// TIA Portal V15 export
// export: Created 2018-05-29T12:25:38.1552518Z, ExportSetting WithDefaults, DisplayName Totally Integrated Automation Portal, DisplayVersion V15, DisplayName STEP 7 Professional, DisplayVersion V15, DisplayName WinCC Professional, DisplayVersion V15, DisplayName TIA Portal Openness, DisplayVersion V15
FUNCTION_BLOCK "EM_I_OUT"   // FB1, STL
TITLE = EM_I_OUT_fc
{ S7_Optimized_Access := 'TRUE' }
VERSION : 0.1
// EM_I_OUT
// stored: AutoNumber true, UDAEnableTagReadback false
   VAR_INPUT
      sampletime : Real;   // the scantime of this EM/phase, used to increase timers
      em_id : Int;   // undefined - undefined
      Request : Int;   // undefined - undefined
      Command : Int;   // undefined - undefined
      Pressure_SP : REAL;   // undefined - undefined
      Pump_RUN : Bool;   // undefined - undefined
      Pump_QERR : BOOL;   // undefined - General Error
      Pump_EERR : BOOL;   // undefined - External Error
      FS01_PV : Bool;   // Flow Switch - Digital Measurement
      PIC01_PV : REAL;   // Pressure Controller - undefined
      PIC01_ERR : BOOL;   // Pressure Controller - undefined
      LT01_PV : Real;   // Level Transmitter (m) - undefined
      LT01_AHH : Bool;   // Level Transmitter (m) - undefined
      LT01_AH : Bool;   // Level Transmitter (m) - undefined
      LT01_AL : Bool;   // Level Transmitter (m) - undefined
      LT01_ALL : Bool;   // Level Transmitter (m) - undefined
      LT01_ERR : BOOL;   // Level Transmitter (m) - undefined
      XV_Bottom_OPN : BOOL;   // Automatic Bottom Valve - undefined
      XV_Bottom_CLS : BOOL;   // Automatic Bottom Valve - undefined
      XV_Bottom_MERR : BOOL;   // Automatic Bottom Valve - undefined
      BV_Bottom_OPN : BOOL;   // Manual Bottom Valve - undefined
      BV_Bottom_CLS : BOOL;   // Manual Bottom Valve - undefined
      BV_Bottom_MERR : BOOL;   // Manual Bottom Valve - undefined
      BV_Tran_M04_OPN : BOOL;   // Trnasfer Valve to M04 - undefined
      BV_Tran_M04_CLS : BOOL;   // Trnasfer Valve to M04 - undefined
      BV_Tran_M04_MERR : BOOL;   // Trnasfer Valve to M04 - undefined
   END_VAR
   VAR_OUTPUT
      steptime_s : Real;   // complete steptime in seconds. same value as the other steptimes
      steptime_m : Real;   // complete steptime in minutes. same value as the other steptimes
      steptime_h : Real;   // complete steptime in hours. same value as the other steptimes
      first_scan : Bool;   // first scan of the step active
      last_scan : Bool;   // last scan of the step active
      error_index_db : Bool;   // em_id doesn't fit in the index db
      Owner : Int;   // undefined - undefined
      Status : Int;   // undefined - undefined
      CM_error : Bool;   // undefined - undefined
      CM_error_no : DINT;   // undefined - undefined
      q_bACTVIE : Bool;   // undefined - undefined
      Level : REAL;   // undefined - undefined
      Pressure : REAL;   // undefined - undefined
      Pump_ON : Bool;   // undefined - Switch Motor ON
      Pump_AUT : Bool;   // undefined - Swtich Motor to AUTO
      PIC01_EXT : Bool;   // Pressure Controller - Switch to External Mode
      PIC01_SP : Real;   // Pressure Controller - Operator Setpoint in Internal Mode
      PIC01_AUT : Bool;   // Pressure Controller - Switch to Auto Mode
      PIC01_VAL_OUT : Real;   // Pressure Controller - Operator Output Value
      PIC01_SET_SP : Bool;   // Pressure Controller - undefined
      PIC01_SET_OUT : Bool;   // Pressure Controller - undefined
      XV_Bottom_CMD : BOOL;   // Automatic Bottom Valve - Auto command from program
      BV_Bottom_CMD : BOOL;   // Manual Bottom Valve - Auto command from program
      BV_Tran_M04_CMD : BOOL;   // Trnasfer Valve to M04 - Auto command from program
   END_VAR
   VAR DB_SPECIFIC
      previous_Command : Int;   // previous Command
      SP_PV : "EM_I_OUT_UDT";   // UDT for receiving Setpoints and sending Process Values
   END_VAR
   VAR_TEMP
      initial_scan : Bool;   // pulse active on the first cycle of a new scan
      T_dbnum : Int;   // DB number of this block
      T_address : Int;   // address in the Index Table DB
      T_length : Int;   // length of the Index Table DB
   END_VAR
BEGIN

NETWORK
TITLE = Publish DB number to EM Index
// The EM will publish its DB number to the EM Index table


//### 0] init
      CLR;
      =     #error_index_db;


//### 1] Check if the ID of this EM fits inside the EM Index table

      OPN   "EM_Index";  //Open data block as shared data block
      L     DBLG;  //Load length of shared data block (length of DB)
      T     #T_length;  //transfer length to length

      L     #T_length;  //length=length/2
      L     2;
      /I;
      T     #T_length;

// Error and end the block if id bigger than length of the DB
      L     #T_length;
      L     #em_id;
      <=D;
      =     #error_index_db;
      BEC;  //if id is bigger than length end the block

//### 2] Write this DB number to the EM Index table

// find the number of the current fb
      L     DINO;
      T     #T_dbnum;  //find the db number of current fb

// calculate the real address
      L     #em_id;
      L     2;
      *I;
      T     #T_address;

// prepare the pointer for the location in the EM Index DB
// todo: can this code not simpeler? Probably no need to add with the zero-pointer
      OPN   "EM_Index";
      L     P#DBX0.0;
      L     #T_address;
      SLD   3;
      +D;
      LAR1;

//write the DB number to the real address
      L     #T_dbnum;
      T     DBW [AR1, P#0.0];





NETWORK
TITLE = Copy all Setpoints from the UDT
// network comment





      L     #SP_PV.Request;
      T     #Request;



      L     #SP_PV.Command;
      T     #Command;



      L     #SP_PV.Pressure_SP;
      T     #Pressure_SP;




NETWORK
TITLE = Acquiring logic
// network comment


      L     #Request;
      T     #Owner;



NETWORK
TITLE = Steptimers
// If the previous Command is not the same as the current one
// then reset the timers, else increase them
// This is at the start of the FB because normal commandchanges will take
// till the next cycle to become active


// check if Command == previous_Command
      L     #Command;
      L     #previous_Command;
      ==I;  //if condition true then {
      JCN   TIM1;

// increase timer
      L     #sampletime;
      L     #steptime_s;
      +R;
      T     #steptime_s;

      JU    TIM2;
TIM1: NOP   0;

// reset timer
      L     0.0;
      T     #steptime_s;

TIM2: NOP   0;  //end if

// calculate the other two timers
      L     #steptime_s;
      L     60.0;
      /R;
      T     #steptime_m;

      L     60.0;
      /R;
      T     #steptime_h;



NETWORK
TITLE = detect initial scan
// create a pulse active on the first cycle of a new scan
// this signal can be used in the state to execute some actions in the first cycle of the state


      L     #Command;
      L     #previous_Command;
      <>I;
      =     #initial_scan;



NETWORK
TITLE = Save old step
// network comment


      L     #Command;
      T     #previous_Command;



NETWORK
TITLE = Collect the errors from the CMs
// network comment


      CLR;
      O     #Pump_QERR;
      O     #Pump_EERR;
      O     #PIC01_ERR;
      O     #LT01_ERR;
      O     #XV_Bottom_MERR;
      O     #BV_Bottom_MERR;
      O     #BV_Tran_M04_MERR;
      =     #CM_error;



NETWORK
TITLE = Assign a message number to each error
// This code tries to assign an error message to each CM error
// If multiple CMs have an error then it only stores one
// This is the EM type so we don't know which CM instance is connected
// So the error only contains the general name of the CM instance
// If the actual name needs to be shown then it could be deducted
// at a higher level using the CM name and EM instance 
// network_end.render(lib, "ssign a message number to each error") }}


      CLR;

// clear the error no
      L     0;
      T     #CM_error_no;



      A     #Pump_QERR;
      JCN   E1;

      L     50;  //'CM error: Pump_QERR'
      T     #CM_error_no;

E1:   NOP   0;

      A     #Pump_EERR;
      JCN   E2;

      L     51;  //'CM error: Pump_EERR'
      T     #CM_error_no;

E2:   NOP   0;

      A     #PIC01_ERR;
      JCN   E3;

      L     52;  //'CM error: PIC01_ERR'
      T     #CM_error_no;

E3:   NOP   0;

      A     #LT01_ERR;
      JCN   E4;

      L     53;  //'CM error: LT01_ERR'
      T     #CM_error_no;

E4:   NOP   0;

      A     #XV_Bottom_MERR;
      JCN   E5;

      L     54;  //'CM error: XV_Bottom_MERR'
      T     #CM_error_no;

E5:   NOP   0;

      A     #BV_Bottom_MERR;
      JCN   E6;

      L     55;  //'CM error: BV_Bottom_MERR'
      T     #CM_error_no;

E6:   NOP   0;

      A     #BV_Tran_M04_MERR;
      JCN   E7;

      L     56;  //'CM error: BV_Tran_M04_MERR'
      T     #CM_error_no;

E7:   NOP   0;



NETWORK
TITLE = START OF THE STATES
// ################################
// ################################
// 	Placeholder network to indicate the start of the actual sequence
// ################################	  
// ################################


// empty placeholder network



NETWORK
TITLE = State 0: undefined


// skip this network if stepnumber not equal to 0
      L     #Command;
      L     0;
      ==I;
      JCN   J1;

//---------------------------------
// Actions (continuous)
//---------------------------------

// Action: stop Pump
      CLR;
      =     #Pump_ON;

// Action: close XV_Bottom
      CLR;
      =     #XV_Bottom_CMD;

// Action: close BV_Bottom
      CLR;
      =     #BV_Bottom_CMD;

// Action: close BV_Tran_M04
      CLR;
      =     #BV_Tran_M04_CMD;
//---------------------------------
// --- CONDITIONS ---
//---------------------------------

// Condition Logic
      SET;  //make sure RLO is high so the state can happen when no conditions present

      A     #XV_Bottom_CLS;  //XV_Bottom close
      A     #BV_Bottom_CLS;  //BV_Bottom close
      A     #BV_Tran_M04_CLS;  //BV_Tran_M04 close
      JCN   L1;

      L     #Command;
      T     #Status;

L1:   NOP   0;

D1:   NOP   0;

//---------------------------------
// End of network: jump here if step not active
// Jump to end of this FB if the step has been active to avoid
// execution of another step in the same scan
//---------------------------------
      JU    ENDS;
J1:   NOP   0;




NETWORK
TITLE = State 1: undefined


// skip this network if stepnumber not equal to 1
      L     #Command;
      L     1;
      ==I;
      JCN   J2;

//---------------------------------
// Actions (continuous)
//---------------------------------

// Action: stop Pump
      CLR;
      =     #Pump_ON;

// Action: open XV_Bottom
      SET;
      =     #XV_Bottom_CMD;
//---------------------------------
// --- CONDITIONS ---
//---------------------------------

// Condition Logic
      SET;  //make sure RLO is high so the state can happen when no conditions present

      A     #XV_Bottom_OPN;  //XV_Bottom open
      JCN   L2;

      L     #Command;
      T     #Status;

L2:   NOP   0;

D2:   NOP   0;

//---------------------------------
// End of network: jump here if step not active
// Jump to end of this FB if the step has been active to avoid
// execution of another step in the same scan
//---------------------------------
      JU    ENDS;
J2:   NOP   0;




NETWORK
TITLE = State 2: undefined


// skip this network if stepnumber not equal to 2
      L     #Command;
      L     2;
      ==I;
      JCN   J3;

//---------------------------------
// Actions (first scan)
//---------------------------------
      A     #initial_scan;
      JCN   C3;
      L     -1.0;  //value to show that the EM is in a state transition
      T     #Status;

// Action: PIC01_SP = 10.0
      L     10.0;
      T     #PIC01_SP;

// Action: PIC01_SET_SP = true
      SET;
      =     #PIC01_SET_SP;

      JU    D3;
C3:   NOP   0;


//---------------------------------
// Actions (continuous)
//---------------------------------

// Action: start Pump
      SET;
      =     #Pump_ON;

// Action: auto 10.0 bar PIC01
      SET;
      =     #PIC01_AUT;

// Action: open XV_Bottom
      SET;
      =     #XV_Bottom_CMD;

// Action: PIC01_SET_SP = false
      CLR;
      =     #PIC01_SET_SP;
//---------------------------------
// --- CONDITIONS ---
//---------------------------------

// Condition Logic
      SET;  //make sure RLO is high so the state can happen when no conditions present

      A     #Pump_RUN;  //Pump start
      A     #XV_Bottom_OPN;  //XV_Bottom open
      JCN   L3;

      L     #Command;
      T     #Status;

L3:   NOP   0;

D3:   NOP   0;

//---------------------------------
// End of network: jump here if step not active
// Jump to end of this FB if the step has been active to avoid
// execution of another step in the same scan
//---------------------------------
      JU    ENDS;
J3:   NOP   0;




NETWORK
TITLE = State 3: undefined


// skip this network if stepnumber not equal to 3
      L     #Command;
      L     3;
      ==I;
      JCN   J4;

//---------------------------------
// Actions (continuous)
//---------------------------------

// Action: stop Pump
      CLR;
      =     #Pump_ON;

// Action: open BV_Bottom
      SET;
      =     #BV_Bottom_CMD;

// Action: open BV_Tran_M04
      SET;
      =     #BV_Tran_M04_CMD;
//---------------------------------
// --- CONDITIONS ---
//---------------------------------

// Condition Logic
      SET;  //make sure RLO is high so the state can happen when no conditions present

      A     #BV_Bottom_OPN;  //BV_Bottom open
      A     #BV_Tran_M04_OPN;  //BV_Tran_M04 open
      JCN   L4;

      L     #Command;
      T     #Status;

L4:   NOP   0;

D4:   NOP   0;

//---------------------------------
// End of network: jump here if step not active
// Jump to end of this FB if the step has been active to avoid
// execution of another step in the same scan
//---------------------------------
      JU    ENDS;
J4:   NOP   0;




NETWORK
TITLE = State 4: undefined


// skip this network if stepnumber not equal to 4
      L     #Command;
      L     4;
      ==I;
      JCN   J5;

//---------------------------------
// Actions (first scan)
//---------------------------------
      A     #initial_scan;
      JCN   C5;
      L     -1.0;  //value to show that the EM is in a state transition
      T     #Status;

// Action: PIC01_SP = Pressure_SP
      L     #Pressure_SP;
      T     #PIC01_SP;

// Action: PIC01_SET_SP = true
      SET;
      =     #PIC01_SET_SP;

      JU    D5;
C5:   NOP   0;


//---------------------------------
// Actions (continuous)
//---------------------------------

// Action: start Pump
      SET;
      =     #Pump_ON;

// Action: auto Pressure_SP PIC01
      SET;
      =     #PIC01_AUT;

// Action: open BV_Bottom
      SET;
      =     #BV_Bottom_CMD;

// Action: open BV_Tran_M04
      SET;
      =     #BV_Tran_M04_CMD;

// Action: PIC01_SET_SP = false
      CLR;
      =     #PIC01_SET_SP;
//---------------------------------
// --- CONDITIONS ---
//---------------------------------

// Condition Logic
      SET;  //make sure RLO is high so the state can happen when no conditions present

      A     #Pump_RUN;  //Pump start
      A     #BV_Bottom_OPN;  //BV_Bottom open
      A     #BV_Tran_M04_OPN;  //BV_Tran_M04 open
      JCN   L5;

      L     #Command;
      T     #Status;

L5:   NOP   0;

D5:   NOP   0;

//---------------------------------
// End of network: jump here if step not active
// Jump to end of this FB if the step has been active to avoid
// execution of another step in the same scan
//---------------------------------
      JU    ENDS;
J5:   NOP   0;




NETWORK
TITLE = State 5: undefined


// skip this network if stepnumber not equal to 5
      L     #Command;
      L     5;
      ==I;
      JCN   J6;

//---------------------------------
// Actions (first scan)
//---------------------------------
      A     #initial_scan;
      JCN   C6;
      L     -1.0;  //value to show that the EM is in a state transition
      T     #Status;

// Action: PIC01_VAL_OUT = 20.0
      L     20.0;
      T     #PIC01_VAL_OUT;

// Action: PIC01_SET_OUT = true
      SET;
      =     #PIC01_SET_OUT;

      JU    D6;
C6:   NOP   0;


//---------------------------------
// Actions (continuous)
//---------------------------------

// Action: start Pump
      SET;
      =     #Pump_ON;

// Action: manual 20.0 Hz PIC01
      CLR;
      =     #PIC01_AUT;

// Action: open XV_Bottom
      SET;
      =     #XV_Bottom_CMD;

// Action: PIC01_SET_OUT = false
      CLR;
      =     #PIC01_SET_OUT;
//---------------------------------
// --- CONDITIONS ---
//---------------------------------

// Condition Logic
      SET;  //make sure RLO is high so the state can happen when no conditions present

      A     #Pump_RUN;  //Pump start
      A     #XV_Bottom_OPN;  //XV_Bottom open
      JCN   L6;

      L     #Command;
      T     #Status;

L6:   NOP   0;

D6:   NOP   0;

//---------------------------------
// End of network: jump here if step not active
// Jump to end of this FB if the step has been active to avoid
// execution of another step in the same scan
//---------------------------------
      JU    ENDS;
J6:   NOP   0;




NETWORK
TITLE = END OF THE STATES
// ################################
// ################################
// 	Placeholder network to indicate the end of the actual sequence
// ################################	  
// ################################


// jump location for the state that is currently active
ENDS: NOP   0;



NETWORK
TITLE = eneral Actions - After
// General Actions - After


// Action: Level = LT01
      L     #LT01_PV;
      T     #Level;

// Action: Pressure = PIC01
      L     #PIC01_PV;
      T     #Pressure;


NETWORK
TITLE = Copy all Process Values to the UDT
// network comment





      L     #Owner;
      T     #SP_PV.Owner;



      L     #Status;
      T     #SP_PV.Status;



      A     #CM_error;
      =     #SP_PV.CM_error;



      L     #CM_error_no;
      T     #SP_PV.CM_error_no;



      A     #q_bACTVIE;
      =     #SP_PV.q_bACTVIE;



      L     #Level;
      T     #SP_PV.Level;



      L     #Pressure;
      T     #SP_PV.Pressure;




NETWORK
TITLE = Clean up request
// Phases don't clean up their requests on the EM side
// So at the end of the EM reset the request
// If the phase is still there then it will write the request again by the next scan


      L     0;
      T     "request";



NETWORK
TITLE = network title
// network comment


// empty placeholder network


END_FUNCTION_BLOCK
